FUNCTION_BLOCK FB_CTRL_PI (* Basic Function Block Type *)
  (* Standard: 61499-2 *)
  (* Version 0.0, 2011-08-25, 4DIAC-IDE, 4DIAC-Consortium *)
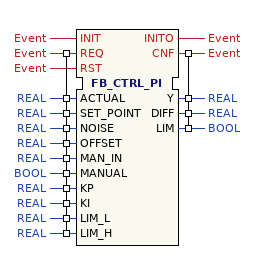
  EVENT_INPUT
    INIT; (* Initialization Request *)
    REQ WITH ACTUAL, SET_POINT, NOISE, OFFSET, MAN_IN, MANUAL, KP, KI, LIM_L, LIM_H; (* Normal Execution Request *)
    RST;
  END_EVENT
  EVENT_OUTPUT
    INITO; (* Initialization Confirm *)
    CNF WITH Y, DIFF, LIM; (* Execution Confirmation *)
  END_EVENT
  VAR_INPUT
    ACTUAL : REAL; (* process value *)
    SET_POINT : REAL; (* setpoint *)
    NOISE : REAL; (* noise reduction *)
    OFFSET : REAL; (* offset for the output *)
    MAN_IN : REAL; (* input value for manual operation *)
    MANUAL : BOOL; (* swithc to manual mode, MAN = TRUE *)
    KP : REAL := 1.0; (* proportional gain of the controller *)
    KI : REAL := 1.0; (* integral gain of the controller *)
    LIM_L : REAL := -1000.0; (* output lower limit *)
    LIM_H : REAL := 1000.0; (* output higher limit *)
  END_VAR
  VAR_OUTPUT
    Y : REAL; (* output of the controller *)
    DIFF : REAL; (* deviation between act and setpoint *)
    LIM : BOOL; (* TRUE if the output has reached a limit *)
  END_VAR
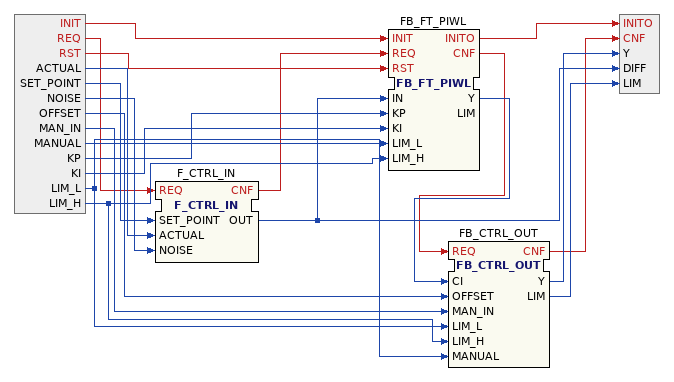
  FBS
    FB_CTRL_OUT : FB_CTRL_OUT;
    FB_FT_PIWL : FB_FT_PIWL;
    F_CTRL_IN : F_CTRL_IN;
  END_FBS
  EVENT_CONNECTIONS
    REQ TO F_CTRL_IN.REQ;
    F_CTRL_IN.CNF TO FB_FT_PIWL.REQ;
    FB_FT_PIWL.CNF TO FB_CTRL_OUT.REQ;
    FB_CTRL_OUT.CNF TO CNF;
    RST TO FB_FT_PIWL.RST;
    INIT TO FB_FT_PIWL.INIT;
    FB_FT_PIWL.INITO TO INITO;
  END_CONNECTIONS
  DATA_CONNECTIONS
    FB_CTRL_OUT.Y TO Y;
    FB_CTRL_OUT.LIM TO LIM;
    FB_FT_PIWL.Y TO FB_CTRL_OUT.CI;
    SET_POINT TO F_CTRL_IN.SET_POINT;
    ACTUAL TO F_CTRL_IN.ACTUAL;
    NOISE TO F_CTRL_IN.NOISE;
    KP TO FB_FT_PIWL.KP;
    KI TO FB_FT_PIWL.KI;
    LIM_L TO FB_FT_PIWL.LIM_L;
    LIM_H TO FB_FT_PIWL.LIM_H;
    LIM_L TO FB_CTRL_OUT.LIM_L;
    LIM_H TO FB_CTRL_OUT.LIM_H;
    MANUAL TO FB_CTRL_OUT.MANUAL;
    MAN_IN TO FB_CTRL_OUT.MAN_IN;
    OFFSET TO FB_CTRL_OUT.OFFSET;
    F_CTRL_IN.OUT TO FB_FT_PIWL.IN;
    F_CTRL_IN.OUT TO DIFF;
  END_CONNECTIONS
END_FUNCTION_BLOCK
